// TwinCAT 3 PLC project Aufgabe1
// ProgramVersion: 3.1.4023.0
// libraries:
//   Tc2_Standard, * (Beckhoff Automation GmbH)
//   Tc2_System, * (Beckhoff Automation GmbH)
//   Tc3_Module, * (Beckhoff Automation GmbH)
// project tree:
//   / FastTask.TcTTO, PlcTask.TcTTO, SlowTask.TcTTO
//   POUs/ FAST.TcPOU, MAIN.TcPOU, SLOW.TcPOU
// real-time tasks:
//   TASK PlcTask: cycle T#1ms, priority 1, ADS port 350
//   TASK FastTask: cycle T#300us, priority 2, ADS port 351
//   TASK SlowTask: cycle T#10ms, priority 3, ADS port 352
//   TASK PlcTask1: cycle T#10ms, priority 20, ADS port 353
// I/O:
//   DEVICE Device 1 (EtherCAT), AmsNetId 10.155.117.35.2.1
//     Term 1 (EK1100) [EK1100 EtherCAT Coupler (2A E-Bus)]
//       Term 2 (EL2004) [EL2004 4Ch. Dig. Output 24V, 0.5A]
//       Term 3 (EL1004) [EL1004 4Ch. Dig. Input 24V, 3ms]
// variable links:
//   Aufgabe3/Aufgabe3 Instance <-> Device 1 (EtherCAT)/Term 1 (EK1100)/Term 2 (EL2004)
//     PlcTask Outputs/GVL_IO.DO_LampGreen <-> Channel 2/Output
//     PlcTask Outputs/GVL_IO.DO_LampOrange <-> Channel 3/Output
//     PlcTask Outputs/GVL_IO.DO_LampRed <-> Channel 1/Output
//   Aufgabe3/Aufgabe3 Instance <-> Device 1 (EtherCAT)/Term 1 (EK1100)/Term 3 (EL1004)
//     PlcTask Inputs/GVL_IO.DI_BtnBlue <-> Channel 2/Input
//     PlcTask Inputs/GVL_IO.DI_BtnGreen <-> Channel 3/Input
//     PlcTask Inputs/GVL_IO.DI_BtnYellow <-> Channel 1/Input

CONFIGURATION Aufgabe1
    RESOURCE PLC ON TwinCAT3
        TASK FastTask(INTERVAL := T#300us, PRIORITY := 2);
        TASK PlcTask(INTERVAL := T#1ms, PRIORITY := 1);
        TASK SlowTask(INTERVAL := T#10ms, PRIORITY := 3);
        PROGRAM FAST WITH FastTask : FAST;
        PROGRAM MAIN WITH PlcTask : MAIN;
        PROGRAM SLOW WITH SlowTask : SLOW;
    END_RESOURCE
END_CONFIGURATION

// ---- POUs/FAST.TcPOU
PROGRAM FAST
VAR
END_VAR

;

END_PROGRAM

// ---- POUs/MAIN.TcPOU
PROGRAM MAIN
VAR
END_VAR

END_PROGRAM

// ---- POUs/SLOW.TcPOU
PROGRAM SLOW
VAR
END_VAR

;

END_PROGRAM
